FUNCTION posicionEstanteria : Array[1..2] of real
VAR_INPUT
END_VAR
VAR
	posicion : ARRAY[1..2] OF REAL;
	// 1 - posicion en X (horizontal)
	// 2 - posicoin en Z (vertical)
	fila: DINT;
	arr2D: INT;
	col: DINT;
END_VAR

FOR fila := 1 TO 6 DO
    FOR col := 1 TO 3 DO
        // la primera posicion libre 
		IF GVLvar.baldasOcupadas[fila,col] = FALSE THEN
			posicionEstanteria := GVLvar.estanteria[fila,col];
			GVLvar.baldasOcupadas[fila,col] := true;
			EXIT;
		END_IF
    END_FOR
END_FOR

END_FUNCTION

(* stored: Version 1.1.0.1, ProductVersion 3.1.4024.15
   POU posicionEstanteria: Id {07b97f28-9015-4126-8fa4-be169375519b}, SpecialFunc None *)
